TYPE ST_TcpCodeReaderParCmd :
STRUCT
    MatchCode : STRING(255);
END_STRUCT
END_TYPE

(* stored: Version 1.1.0.1, ProductVersion 3.1.4024.12
   DUT ST_TcpCodeReaderParCmd: Id {d07bbb25-3c38-412e-90bb-ab8ed174f0f7} *)
